FUNCTION_BLOCK FeedReactorLogic_HMI (* Service Interface Function Block Type *)
  (* Standard: 61499-2 *)
  (* Version 1.0, 10/1/2026, Claude/Hidryco, Schneider Electric, Rev1 - PUMP_PAR (Cmin, T_C2, T_C3, T_FlowLL, capacidade teorica) e PUMP_STS (status das bombas para o simbolo) *)
  PACKAGE SE.Nereda;
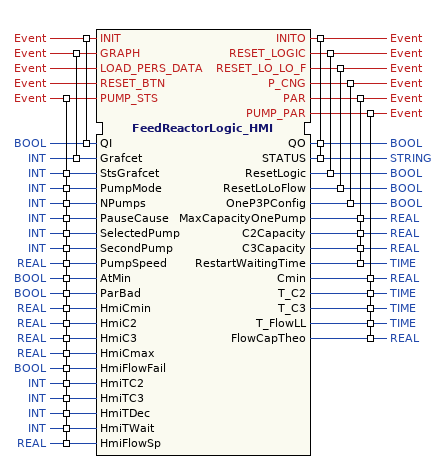
  EVENT_INPUT
    INIT WITH QI;
    GRAPH WITH Grafcet;
    LOAD_PERS_DATA;
    RESET_BTN;
    PUMP_STS WITH StsGrafcet, PumpMode, NPumps, PauseCause, SelectedPump, SecondPump, PumpSpeed, AtMin, ParBad, HmiCmin, HmiC2, HmiC3, HmiCmax, HmiFlowFail, HmiTC2, HmiTC3, HmiTDec, HmiTWait, HmiFlowSp; (* Status das bombas de alimentacao *)
  END_EVENT
  EVENT_OUTPUT
    INITO WITH QO, STATUS;
    RESET_LOGIC WITH ResetLogic;
    RESET_LO_LO_F WITH ResetLoLoFlow;
    P_CNG WITH OneP3PConfig;
    PAR WITH MaxCapacityOnePump, C2Capacity, C3Capacity, RestartWaitingTime;
    PUMP_PAR WITH Cmin, T_C2, T_C3, T_FlowLL, FlowCapTheo; (* Parametros das bombas (Cmin, tempos, capacidade teorica) *)
  END_EVENT
  VAR_INPUT
    QI : BOOL;
    Grafcet : INT;
    StsGrafcet : INT;
    PumpMode : INT;
    NPumps : INT;
    PauseCause : INT;
    SelectedPump : INT;
    SecondPump : INT;
    PumpSpeed : REAL;
    AtMin : BOOL;
    ParBad : BOOL;
    HmiCmin : REAL;
    HmiC2 : REAL;
    HmiC3 : REAL;
    HmiCmax : REAL;
    HmiFlowFail : BOOL;
    HmiTC2 : INT;
    HmiTC3 : INT;
    HmiTDec : INT;
    HmiTWait : INT;
    HmiFlowSp : REAL;
  END_VAR
  VAR_OUTPUT
    QO : BOOL; (* Event Output Qualifier *)
    STATUS : STRING; (* Service Status *)
    ResetLogic : BOOL;
    ResetLoLoFlow : BOOL;
    OneP3PConfig : BOOL; (* = FALSE : One Pump | = TRUE : 3 Pumps *)
    MaxCapacityOnePump : REAL; (* Cmax: velocidade de 1 bomba acima da qual entra a 2a [% velocidade] *)
    C2Capacity : REAL; (* C2: velocidade das bombas na entrada de uma nova bomba [% velocidade] *)
    C3Capacity : REAL; (* C3: velocidade das 2 bombas abaixo da qual sai 1 [% velocidade] *)
    RestartWaitingTime : TIME; (* Tempo de espera para retomar a alimentacao (pH/condutividade/vazao LL) *)
    Cmin : REAL; (* Velocidade minima de cada bomba em servico [% velocidade] *)
    T_C2 : TIME; (* Tempo com as bombas em C2 *)
    T_C3 : TIME; (* Tempo abaixo de C3 para retirar 1 bomba *)
    T_FlowLL : TIME; (* Vazao LL do 40FT0003 com bomba rodando por este tempo = para a alimentacao (0 = desabilitado) *)
    FlowCapTheo : REAL; (* Capacidade teorica de 1 bomba a 100 % [m3/h] (falha do medidor; 0 = usa a faixa do medidor) *)
  END_VAR
  SERVICE /
    SEQUENCE 
    END_SEQUENCE
  END_SERVICE
END_FUNCTION_BLOCK
